// TIA Portal V20 export
TYPE "UDT_OPC_TaughtPositionsItems"
   STRUCT
      StationNumber : Byte;
      AxisId : DInt;
      PositionId : DInt;
      Value : LReal;
   END_STRUCT;
END_TYPE
